FUNCTION_BLOCK TcoDataman_v_5_x_xTests EXTENDS TcoCore._internals_TcoContext
VAR
//	{attribute addProperty Name "<#Dataman 260#>"}
	_dm260 : TcoCognexVision.TcoDataman_v_5_x_x(THIS^);
//	{attribute addProperty Name "<#Dataman 8700#>"}
	_dm8700 : TcoCognexVision.TcoDataman_v_5_x_x(THIS^);
END_VAR

METHOD PROTECTED Main
THIS^.Environment.Messaging.MinLevel := eMessageCategory.Trace;

_dm8700.Config.ContinuousReading := TRUE;

_dm260(inoIoData:= IO.dm260);
_dm8700(inoIoData:= IO.dm8700);

_dm260.Service();
_dm8700.Service();
END_METHOD

END_FUNCTION_BLOCK

(* stored: Version 1.1.0.1, ProductVersion 3.1.4024.11
   POU TcoDataman_v_5_x_xTests: Id {802c992c-138b-01dc-1d08-36966d5f7699}, SpecialFunc None
   Method Main: Id {48e4cb4c-415e-0c4b-094e-2037721a0dd2} *)
